{attribute addProperty BoxType "EK1100-0000-0018"}
{attribute addProperty Id "Beckhoff_ELM9xxxEK1122Beckhoff_ELM9xxxEK1122_E008DD2D162A_0002_ELM9410_0000_0016ELM9410_5F7BBEA262578.125A_0003_ELM9410_0000_0017ELM9410_5F7BBEA262578.125A_0004_ELM9410_0000_0018ELM9410_75EA563B52065A_0005_ELM9410_0000_0019ELM9410_75EA563B52065A_0006_ELM9410_0000_0020ELM9410_75EA563B52065"}
{attribute addProperty CRC "130271166"}
{attribute addProperty SizeInBites "2826"}
{attribute addProperty SizeInBytes "353.25"}
TYPE Beckhoff_ELM9xxx_07C3C7BE EXTENDS EK1100_179A0949 :
STRUCT
	{attribute addProperty Name "Beckhoff_ELM9xxxEK1122"}
	Beckhoff_ELM9xxxEK1122 : Beckhoff_ELM9xxxEK1122_E008DD2D;
	{attribute addProperty Name "A_0002_ELM9410_0000_0016"}
	A_0002_ELM9410_0000_0016 : ELM9410_5F7BBEA2;
	{attribute addProperty Name "A_0003_ELM9410_0000_0017"}
	A_0003_ELM9410_0000_0017 : ELM9410_5F7BBEA2;
	{attribute addProperty Name "A_0004_ELM9410_0000_0018"}
	A_0004_ELM9410_0000_0018 : ELM9410_75EA563B;
	{attribute addProperty Name "A_0005_ELM9410_0000_0019"}
	A_0005_ELM9410_0000_0019 : ELM9410_75EA563B;
	{attribute addProperty Name "A_0006_ELM9410_0000_0020"}
	A_0006_ELM9410_0000_0020 : ELM9410_75EA563B;
END_STRUCT
END_TYPE

(* stored: Version 1.2.0.0, ProductVersion 3.1.4024.9
   DUT Beckhoff_ELM9xxx_07C3C7BE: Id {ae93174f-6975-4df9-9d65-bf178697c4a3} *)
